// Digital output interface
INTERFACE I_DigitalOut EXTENDS I_DIO

// Returns the blinking period
PROPERTY BlinkPeriod : TIME
GET
END_GET
END_PROPERTY

// Get the command issued to the digital output
PROPERTY Command : E_DOCommand
GET
END_GET
END_PROPERTY

// Set the direct control value
PROPERTY DirectControl : BOOL
SET
END_SET
END_PROPERTY

// Returns the flash time
PROPERTY FlashTime : TIME
GET
END_GET
END_PROPERTY

// Get HMI data
PROPERTY HmiData : ST_HmiDigitalOut
GET
END_GET
END_PROPERTY

// Set the square wave period when blinking (default 2s)
METHOD SetBlinkPeriod
VAR_INPUT
	tPeriod		: TIME;			// Blink period
END_VAR
END_METHOD

// Set digital output command
METHOD SetCommand
VAR_INPUT
	eCommandIn		: E_DOCommand;		// Command
END_VAR
END_METHOD

// Set the time to toggle the output when flashing (default 2s)
METHOD SetFlashTime
VAR_INPUT
	tTime		: TIME;			// Flash time
END_VAR
END_METHOD

// Get the digital output state (enum)
PROPERTY State : E_DOState
GET
END_GET
END_PROPERTY

// Get the digital output boolean value
PROPERTY Value : BOOL
GET
END_GET
END_PROPERTY

END_INTERFACE

(* stored: Version 1.1.0.1, ProductVersion 3.1.4024.12
   Itf I_DigitalOut: Id {cf107e87-cae7-441e-b181-1e390d075020}
   Folder Methods: Id {c9efb76e-7a74-4d7c-8a84-00d77b8d4848}
   Folder Properties: Id {23ef8473-f8ea-49f3-bab8-e3e7b7970758}
   Property BlinkPeriod: Id {1bc11fdd-6b92-463a-98c1-4da471c4d7a0}
   Get Get: Id {dd3ced2b-a83f-4528-9f9f-bc0ff7f263cf}
   Property Command: Id {aec988b8-6d95-4cc4-9c6c-5d8817e4adac}
   Get Get: Id {75ef1f63-adfa-4658-bc09-37eb2bb99450}
   Property DirectControl: Id {6b8d967a-0d66-4223-bc69-b45f8a29e9e1}
   Set Set: Id {48c4bdcb-84d3-40b5-a73b-4751b7c90a28}
   Property FlashTime: Id {721f5d0d-a5c6-48d4-96ad-09a937b1da6f}
   Get Get: Id {c9add764-0bf7-48b2-9684-7ecc5438e950}
   Property HmiData: Id {a7db2afb-0f4e-4e64-8fd5-b37821d84e96}
   Get Get: Id {295e0afa-6f74-4b5e-a336-5ed745c05fd7}
   Method SetBlinkPeriod: Id {b6226cba-f933-4d83-bd14-6c57f5441b9a}
   Method SetCommand: Id {4df4f8c7-9458-4f8d-92e5-f547dafec721}
   Method SetFlashTime: Id {b7750966-a6db-4aa4-b9d9-f203c11bb7a4}
   Property State: Id {a6795d43-60ae-433b-b885-aa638e2a8062}
   Get Get: Id {1aea6945-a74a-4ebb-8a26-cd7085efddbb}
   Property Value: Id {432140b8-af35-4b76-a181-da322f7077fa}
   Get Get: Id {06fd0cad-e0e7-40b1-b6fd-3596ec1f088e} *)
